Yaskawa INFORM job: TEST04072.JBI

/JOB
//NAME TEST04072
//POS
///NPOS 3,0,0,0,0,0
///TOOL 0
///POSTYPE PULSE
///PULSE
C00000=0,1,-6,-2,-1,-2
C00001=28866,77748,22500,-3,10037,-2
C00002=-53005,77160,22540,-2,10662,-2
//INST
///DATE 2016/07/05 16:46
///ATTR SC,RW
///GROUP1 RB1
NOP
MOVJ C00000 VJ=10.00
MOVJ C00001 VJ=10.00
DOUT OT#(1) ON
MOVJ C00002 VJ=5.00
DOUT OT#(1) OFF
END
